(* PLC project AcquisitionStaging.project, CODESYS CODESYS V3.5 SP19 Patch 1 *)
(* stored: creationDateTime 2026-08-02T00:00:00, modificationDateTime 2026-08-02T00:00:00 *)

PROGRAM PRG_02_Acquisition_Staging_CFC
  VAR
    instResetAggregation : FB_ResetAggregation;
    instAcquisitionRouter : FB_AcquisitionRouter;
  END_VAR
  VAR_OUTPUT
    CmdReset : ST_ResetCommand;
    HwIn : ST_HardwareImage;
    WinchInputSourceChanged : BOOL;
  END_VAR

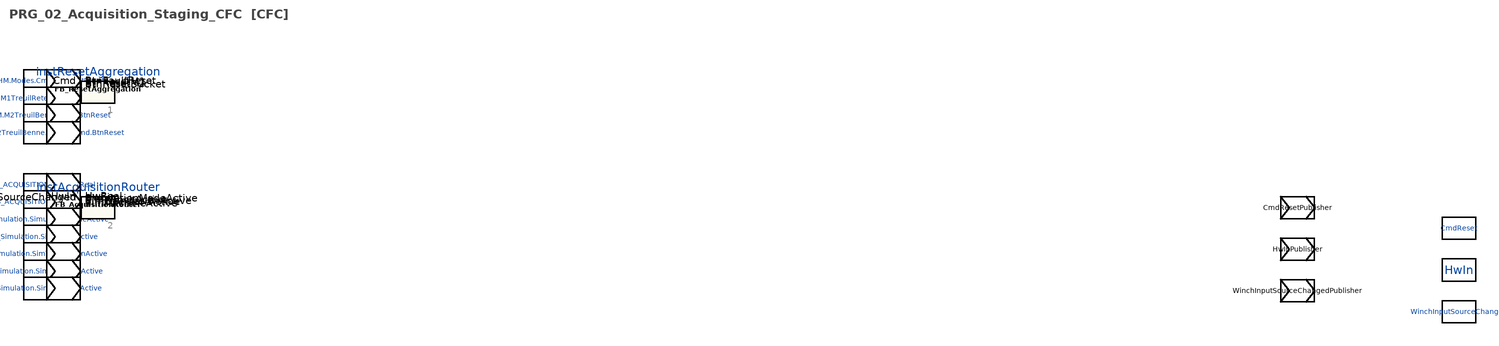
(* CFC diagram, written out as Structured Text *)
instResetAggregation(BtnFaultReset := GVL_IHM.Modes.Cmd.BtnFaultReset, BtnResetM1 := GVL_IHM.M1TreuilRetenue.Cmd.BtnReset, BtnResetM2 := GVL_IHM.M2TreuilBenne.Cmd.BtnReset, BtnResetBucket := GVL_IHM.M2TreuilBenne.Bucket.Cmd.BtnReset);
instAcquisitionRouter(HwReal := PRG_ACQUISITION_CFC.HwReal, HwSim := PRG_ACQUISITION_CFC.HwSim, SimulationModeActive := GVL_Simulation.SimulationModeActive, SimWinchActive := GVL_Simulation.SimWinchActive, SimTranslationActive := GVL_Simulation.SimTranslationActive, SimOperatorActive := GVL_Simulation.SimOperatorActive, SimMachineActive := GVL_Simulation.SimMachineActive);
CmdReset := instResetAggregation.Cmd;
HwIn := instAcquisitionRouter.HwIn;
WinchInputSourceChanged := instAcquisitionRouter.WinchInputSourceChanged;
END_PROGRAM
